FUNCTION FC_LrealFormatter : T_SHORT_STR
VAR_INPUT
	iLreal:				LREAL;
	iNumberOfDecimals:	INT;
END_VAR

FC_LrealFormatter := LREAL_TO_FMTSTR(in := iLreal, iPrecision := iNumberOfDecimals, bRound := FALSE);

END_FUNCTION

(* stored: Version 1.1.0.1, ProductVersion 3.1.4026.18
   POU FC_LrealFormatter: Id {f5832aa7-957a-410a-a98c-fc99a6ce302f}, SpecialFunc None *)
